PROGRAM MAIN
VAR
	fbValveHotWater:	FB_Valve;
	fbValveColdWater:	FB_Valve;
	fbValveBypass:		FB_Valve;
	bValve:		BOOL;
END_VAR

fbValveHotWater(bIn:=TRUE, bOut=>bValve);

END_PROGRAM

(* stored: Version 1.1.0.1
   POU MAIN: Id {6dbe50d1-c61c-4b3b-8c13-53fcd0f25ec9}, SpecialFunc None *)
